PROGRAM prgCalc
VAR
	fbQ56Counter	: FB_EnergyCounter;
	lrPowerQ56		: LREAL;						//{#lynus.ag#()}
END_VAR
VAR PERSISTENT
	lrCounterQ56	: LREAL;						//{#lynus.ag#()}
	lrCO2Enphase	: LREAL;						//{#lynus.ag#()}
	lrCO2PV			: LREAL;						//{#lynus.ag#()}
END_VAR

// calc Output 5 & 6, 230V 16A, Schuko
// choose one of the two calc-options

// 1 -- if prgPV is in use
// lrPowerQ56 := (prgEM.lrPowerEM1 + prgBattery.lrPowerBatt + prgPV.lrPowerPV) - (prgEM.lrPowerEM2 + prgEM.lrPowerEM3 + prgEM.lrPowerEM4 + prgCS.lrPowerCS);
lrPowerQ56 := LIMIT(0,(prgEM.lrPowerEM1) - (prgEM.lrPowerEM2 + prgEM.lrPowerEM3 + prgEM.lrPowerEM4 + prgCS.lrPowerCS),10);

// 2 -- if prgEnphase is in use
// lrPowerQ56 := (prgEM.lrPowerEM1 + prgBattery.lrPowerBatt + prgEnphase.lrPowerPV) - (prgEM.lrPowerEM2 + prgEM.lrPowerEM3 + prgEM.lrPowerEM4 + prgCS.lrPowerCS);

fbQ56Counter(
	byActiveTariff:= 1, 
	lrPowerInput:= lrPowerQ56, 
	lrTotalCounterEnergy_Consumption=> , 
	lrTotalCounterEnergy_Production=> , 
	lrCounterEnergyT1_Consumption=> , 
	lrCounterEnergyT2_Consumption=> , 
	lrCounterEnergyT1_Production=> , 
	lrCounterEnergyT2_Production=> );
	
IF fbQ56Counter.lrTotalCounterEnergy_Consumption > lrCounterQ56 THEN  	
	lrCounterQ56 := fbQ56Counter.lrTotalCounterEnergy_Consumption;
END_IF

// calc saved CO2
// lrCO2Enphase := prgEnphase.lrCounterPV * 0.428;
lrCO2PV := prgPV.lrCounterPV * 0.428;

END_PROGRAM

(* stored: Version 1.1.0.1, ProductVersion 3.1.4024.11
   POU prgCalc: Id {8f293646-b958-4b3c-a62b-c5b5b0996568}, SpecialFunc None *)
